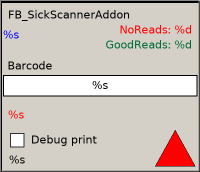
VISUALIZATION V_SickScannerAddon  // 200x172
VAR_IN_OUT
	{attribute 'VAR_IN_OUT_AS_POINTER'}
	fbFunction		: FB_SickScannerAddon;
END_VAR
    Rectangle (0,1 200x171)
    Rectangle (6,150 143x20), "%s", text variable: fbFunction.ConfigFunction.FunctionName
    Label (5,5 139x20), "FB_SickScannerAddon"
    Rectangle (0,25 99x20), "%s", text variable: fbFunction.BaseFunctionData.State.eState
    Rectangle (3,75 194x21), "%s", text variable: fbFunction.BaseFunctionData.LabelData.Label
    Polygon (155,166) (175,130) (195,166) (185,166) (165,166), invisible if: fbFunction.FunctionData.ErrorData.ErrorState = E_ErrorState.OPERATIONAL
    Rectangle (95,35 100x20), "GoodReads: %d", tooltip "good read counter", text variable: fbFunction.FunctionData.AddOnData.Counter[1]
    Rectangle (95,20 100x20), "NoReads: %d", tooltip "no read counter", text variable: fbFunction.FunctionData.AddOnData.Counter[2]
    Rectangle (5,105 192x20), "%s", tooltip "%s", text variable: fbFunction.FunctionData.ErrorData.Error.ErrorCode.Conv, invisible if: fbFunction.FunctionData.ErrorData.Error.ErrorCode.Conv = 0
        p4168582468: fbFunction.FunctionData.ErrorData.Error.ErrorParam
    Label (4,51 52x30), "Barcode"
    Checkbox (8,129 97x22), "Debug print", variable: fbFunction.BaseFunctionData.LabelData.DebugPrint
END_VISUALIZATION

(* stored: Version 1.1.0.1, ProductVersion 3.1.4024.9
   Visu V_SickScannerAddon: Id {983455d3-b49f-40f0-9497-c523d7ace0ca} *)
